{attribute 'qualified_only'}
{attribute 'strict'}
TYPE E_AXIS_STATE :
(
	uninit:=0,
	opening,
	open_dec,
	opened,
	closing,
	close_dec,
	closed,
	ready,
	error
);
END_TYPE

(* stored: Version 1.1.0.1, ProductVersion 3.1.4024.12
   DUT E_AXIS_STATE: Id {7f491dc2-1e1e-47c3-a83e-77e5ec6f7938} *)
